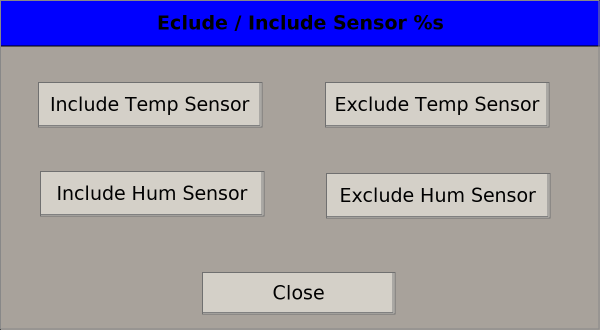
VISUALIZATION Dialog_THT_Field  // 600x330
VAR_IN_OUT
	sHeader : STRING;
	bSetTempIncluded : BOOL;
	bSetHumIncluded : BOOL;
	bSetTempExcluded : BOOL;
	bSetHumExcluded : BOOL;
END_VAR
    Rectangle (0,0 601x46), "Eclude / Include Sensor %s", text variable: sHeader
    Button (38,82 224x45), "Include Temp Sensor"
        OnMouseClick: execute { bSetTempIncluded:= TRUE; }
        OnMouseClick: CloseDialog Dialog=Dialog_CRAH, Result=OK, NumpadKeypadSet=True
    Button (40,171 224x45), "Include Hum Sensor"
        OnMouseClick: execute { bSetHumIncluded:= TRUE; }
        OnMouseClick: CloseDialog Dialog=Dialog_CRAH, Result=OK, NumpadKeypadSet=True
    Button (325,82 224x45), "Exclude Temp Sensor"
        OnMouseClick: execute { bSetTempExcluded:= TRUE; }
        OnMouseClick: CloseDialog Dialog=Dialog_CRAH, Result=OK, NumpadKeypadSet=True
    Button (326,173 224x45), "Exclude Hum Sensor"
        OnMouseClick: execute { bSetHumExcluded:= TRUE; }
        OnMouseClick: CloseDialog Dialog=Dialog_CRAH, Result=OK, NumpadKeypadSet=True
    Button (202,272 193x42), "Close"
        OnMouseClick: CloseDialog Dialog=Dialog_CRAH, Result=OK, NumpadKeypadSet=True
    Line (600,0) (600,330)
    Line (0,330) (600,330)
    Line (0,0) (0,330)
    Line (0,0) (600,0)
END_VISUALIZATION

(* stored: Version 1.1.0.1, ProductVersion 3.1.4024.12
   Visu Dialog_THT_Field: Id {693e1418-c1d0-44ab-878a-ac622a2b02ab} *)
